FUNCTION_BLOCK TransitionList
VAR
	_transition : REFERENCE TO Transition;
	_next : REFERENCE TO TransitionList;
END_VAR

METHOD FB_init : BOOL
VAR_INPUT
	bInitRetains : BOOL; // if TRUE, the retain variables are initialized (warm start / cold start)
	bInCopyCode : BOOL;  // if TRUE, the instance afterwards gets moved into the copy code (online change)
	transition : REFERENCE TO Transition;
	next : REFERENCE TO TransitionList;
END_VAR
IF __ISVALIDREF(transition) THEN
	_transition REF= transition;
END_IF

IF __ISVALIDREF(next) THEN
	_next REF= next;
END_IF
END_METHOD

PROPERTY HasNext : BOOL
GET
HasNext := __ISVALIDREF(_next);
END_GET
END_PROPERTY

PROPERTY Next : REFERENCE TO TransitionList
GET
IF HasNext THEN
	Next REF= _next;
ELSE
	Next REF= 0;
END_IF
END_GET
END_PROPERTY

PROPERTY Value : REFERENCE TO Transition
GET
IF __ISVALIDREF(_transition) THEN
	Value REF= _transition;
ELSE
	Value REF= 0;
END_IF
END_GET
END_PROPERTY

END_FUNCTION_BLOCK

(* stored: Version 1.1.0.1, ProductVersion 3.1.4024.12
   POU TransitionList: Id {10710ab3-1a18-0405-2905-634af37d2937}, SpecialFunc None
   Method FB_init: Id {c00e1da8-e74a-0e15-1ae8-63d2ded94a9d}
   Property HasNext: Id {43ed9a79-3f32-0f0e-1836-960b2b9b4096}
   Get Get: Id {252b315d-3b84-0d3d-2309-00a8b4f35879}
   Property Next: Id {ac24626f-556b-0ebd-00db-32d0c87cb410}
   Get Get: Id {0b61a511-38b4-0f52-0710-f04027b5e534}
   Property Value: Id {eb54e75a-e298-046f-1898-eee9ca8e944c}
   Get Get: Id {66ca52f1-7435-09ad-1a58-c9fac039412a} *)
